(* PLC project  *)

CONFIGURATION EL1918
END_CONFIGURATION
